// Mitsubishi GX Works2 project: 신호등 횡단보도   PLC: Q02/Q02H

PROGRAM MAIN
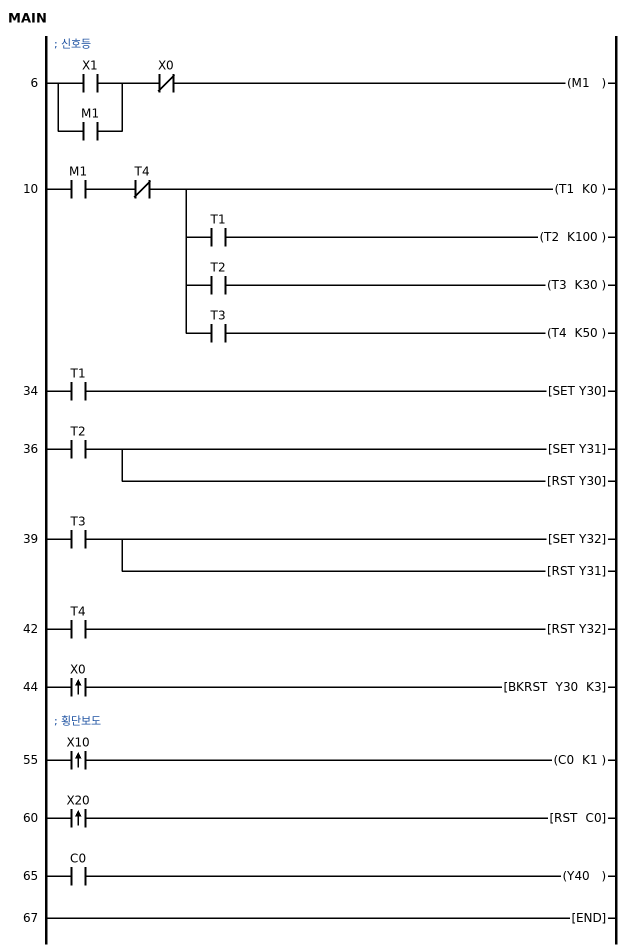
; 신호등
6     LD      X1
      OR      M1
      ANI     X0
      OUT     M1
10    LD      M1
      ANI     T4
      OUT     T1 K0
      MPS
      AND     T1
      OUT     T2 K100
      MRD
      AND     T2
      OUT     T3 K30
      MPP
      AND     T3
      OUT     T4 K50
34    LD      T1
      SET     Y30
36    LD      T2
      SET     Y31
      RST     Y30
39    LD      T3
      SET     Y32
      RST     Y31
42    LD      T4
      RST     Y32
44    LDP     X0
      BKRST   Y30 K3
; 횡단보도
55    LDP     X10
      OUT     C0 K1
60    LDP     X20
      RST     C0
65    LD      C0
      OUT     Y40
67    END
END_PROGRAM
